// TIA Portal V17 export
// export: Created 2025-03-07T09:23:40.9720653Z, ExportSetting WithDefaults, DisplayName Totally Integrated Automation Portal, DisplayVersion V17 Update 8, DisplayName TIA Portal Openness, DisplayVersion V17 Update 8, DisplayName TIA Portal Version Control Interface, DisplayVersion V17, DisplayName SINAMICS Startdrive Advanced, DisplayVersion V17 SP2, DisplayName SINAMICS Startdrive G110M, G120, G120C, G120D, G120P, G115D, DisplayVersion V17 SP2, DisplayName SINAMICS Startdrive G130, G150, S120, S150, SINAMICS MV, S210, DisplayVersion V17 SP2, DisplayName STEP 7 Professional, DisplayVersion V17 Update 8, DisplayName SINUMERIK ONE STEP 7 Toolbox, DisplayVersion V17 Update 12, DisplayName SINUMERIK 840D sl STEP 7 Toolbox, DisplayVersion V17 Update 12, DisplayName STEP 7 Safety, DisplayVersion V17 Update 6, DisplayName WinCC Advanced, DisplayVersion V17 Update 8
DATA_BLOCK "DB2130_TIMERS"   // DB2130
{ S7_Optimized_Access := 'FALSE'; DB_Accessible_From_OPC_UA := 'FALSE' }
AUTHOR : ETXETAR
VERSION : 1.0
// stored: AutoNumber false, DBAccessibleFromOPCUA false, DBAccessibleFromWebserver true, IsOnlyStoredInLoadMemory false, IsWriteProtectedInAS false
   VAR
      TIMER_CH2_ACK_M50 { S7_SetPoint := 'True'} : IEC_TIMER;   // CHANNEL 2 ACKNOWLEDGE M50 TIMER
      TIMER_CH2_ACK_M51 { S7_SetPoint := 'True'} : IEC_TIMER;   // CHANNEL 2 ACKNOWLEDGE M51 TIMER
      TIMER_CH2_ACK_M160 { S7_SetPoint := 'True'} : IEC_TIMER;   // CHANNEL 2 ACKNOWLEDGE M160 TIMER
      TIMER_CH3_ACK_M50 { S7_SetPoint := 'True'} : IEC_TIMER;   // CHANNEL 3 ACKNOWLEDGE M50 TIMER
      TIMER_CH3_ACK_M51 { S7_SetPoint := 'True'} : IEC_TIMER;   // CHANNEL 3 ACKNOWLEDGE M51 TIMER
      TIMER_CH3_ACK_M160 { S7_SetPoint := 'True'} : IEC_TIMER;   // CHANNEL 3 ACKNOWLEDGE M160 TIMER
   END_VAR
BEGIN
   TIMER_CH2_ACK_M50.PT := T#2s;
   TIMER_CH2_ACK_M51.PT := T#2s;
   TIMER_CH2_ACK_M160.PT := T#1s;
   TIMER_CH3_ACK_M50.PT := T#2s;
   TIMER_CH3_ACK_M51.PT := T#2s;
   TIMER_CH3_ACK_M160.PT := T#1s;
END_DATA_BLOCK
